Fanuc KAREL source: CREATE_TPE.kl

PROGRAM T
%NOLOCKGROUP
VAR
 v0 : STRING[40]
 v1 : INTEGER
 v2 : INTEGER
BEGIN
 CREATE_TPE(v0, v1, v2)
END T
